(* IEC 61131-3 sources: learning-path/05_introduction_to_st/src, 2 files *)

(* ---- TankFb.st ---- *)
    FUNCTION_BLOCK Tank
        VAR_INPUT
            cmdFill : BOOL; // Inlet valve is open
            cmdEmptying : BOOL; // Outlet valve is open
            cmdFlush : BOOL; // Inlet and outlet valve is open
            volume : LREAL;
        END_VAR
        VAR_IN_OUT
            inletValve : Valve;
            outletValve : Valve;
        END_VAR
        ;
    END_FUNCTION_BLOCK

(* ---- ExampleProgram.st ---- *)
PROGRAM ExampleProgram
    VAR_EXTERNAL
        //global  variables / instances from the configuration
    END_VAR

    VAR
        // program local variables / instances (static)
    END_VAR

    VAR_TEMP
        // temporary local variables (will be reset in each cycle)
    END_VAR

    ; // program code
END_PROGRAM
